# EPICS autosave request: support/pilatus/1-6/pilatusApp/Db/pilatusROI_N_settings.req
$(DET)ROI$(N)XMin
$(DET)ROI$(N)XMax
$(DET)ROI$(N)YMin
$(DET)ROI$(N)YMax
$(DET)ROI$(N)BgdWidth
$(DET)ROI$(N)Label
